// TIA Portal project "tasl1" (V16)
// Vorlageprojekt für das Buch mit Zielsystem S7-1200

(* hardware
DEVICE "S7-1200-Station_1"  S7-1200 Station
   slot 0: "Baugruppenträger_0"  Rack  V1.0
   slot 1: "PLC_1"  CPU 1211C DC/DC/DC  6ES7 211-1AE40-0XB0  V4.1
*)

// ===== PLC "PLC_1"  CPU 1211C DC/DC/DC =====

VAR_GLOBAL   // PLC tag table "Standard-Variablentabelle"
   "Tag_1" AT %A0.0 : Bool;
   "Tag_2" AT %E0.0 : Bool;
   "Tag_3" AT %E0.1 : Bool;
   "start" AT %I10.0 : Bool;
   "conv6" AT %Q10.0 : Bool;
   "stop" AT %I10.1 : Bool;
   "Tag_7" AT %I10.2 : Bool;
   "pusher" AT %Q10.2 : Bool;
   "Tag_9" AT %M0.0 : Bool;
   "x" AT %M0.1 : Bool;
   "front" AT %I10.4 : Bool;
   "back" AT %I10.3 : Bool;
   "conv2" AT %Q10.1 : Bool;
   "back(1)" AT %I10.3 : Bool;
END_VAR

// folder: System blocks/Program resources

DATA_BLOCK "time"   // DB1
{ S7_Optimized_Access := 'TRUE' }
AUTHOR : Simatic
FAMILY : IEC
NAME : IEC_TMR
VERSION : 1.0
// stored: InstanceOfName IEC_TIMER
"IEC_TIMER"
BEGIN
END_DATA_BLOCK

// folder: (top level)

FUNCTION "MHJ-PLC-Lab-Function-S71200" : Void   // FC9000, SCL
{ S7_Optimized_Access := 'TRUE' }
VERSION : 0.1
   VAR_TEMP
      rdTimeReturn : Int;
      outputTime : DTL;
      SyncVal : Byte;
      forVal : Int;
      forVal_2 : Int;
      Value : Byte;
   END_VAR
   VAR CONSTANT
      CompVal : Byte := 16#34;
      Value_01 : Byte := 16#11;
      Value_01_DW : DWord := 16#A165_D992;
      Value_02_DW : DWord := 16#58BE_4401;
   END_VAR
BEGIN

   #Value:=PEEK(area := 16#82,
        dbNumber := 0,
        byteOffset := 511);
   #Value := #Value + 1;

   POKE(area := 16#82,
        dbNumber := 0,
        byteOffset := 511,
        value := #Value);

   POKE(area:=16#81,
        dbNumber:=0,
        byteOffset:=1016,
        value:=#Value_01_DW);
   POKE(area := 16#81,
        dbNumber := 0,
        byteOffset := 1020,
        value := #Value_02_DW);

   POKE(area := 16#81,
        dbNumber := 0,
        byteOffset := 511,
        value := B#16#00);

   FOR #forVal := 0 TO 120 DO
       FOR #forVal_2:=0 TO 10 DO
           #rdTimeReturn:=RD_SYS_T(#outputTime);
           #rdTimeReturn := WR_SYS_T(#outputTime);
           #rdTimeReturn := RD_SYS_T(#outputTime);
           #rdTimeReturn := WR_SYS_T(#outputTime);
       END_FOR;
       #SyncVal:= PEEK(area := 16#81,
                      dbNumber := 0,
                      byteOffset := 511);
       IF #SyncVal = #CompVal THEN
          GOTO M_1;
       END_IF;
   END_FOR;
   RETURN;

   M_1:
   POKE(area := 16#81,
        dbNumber := 0,
        byteOffset := 511,
        value := B#16#0);
END_FUNCTION

ORGANIZATION_BLOCK "Main"   // OB1, LAD, ProgramCycle
TITLE = "Main Program Sweep (Cycle)"
{ S7_Optimized_Access := 'TRUE' }
VERSION : 0.1
   VAR_INPUT
      Initial_Call : Bool;   // Initial call of this OB
      Remanence : Bool;   // =True, if remanent data are available
   END_VAR
   VAR_TEMP   // added for the SCL form of the ladder/FBD networks
      _w1 : Bool;
   END_VAR
BEGIN

REGION Network 1: Konnektierungsbaustein für PLC-Lab
   // Im Netzwerk 1 wird der Konnektierungsbaustein für PLC-Lab aufgerufen.
   // Dieser Aufruf darf nicht entfernt werden!
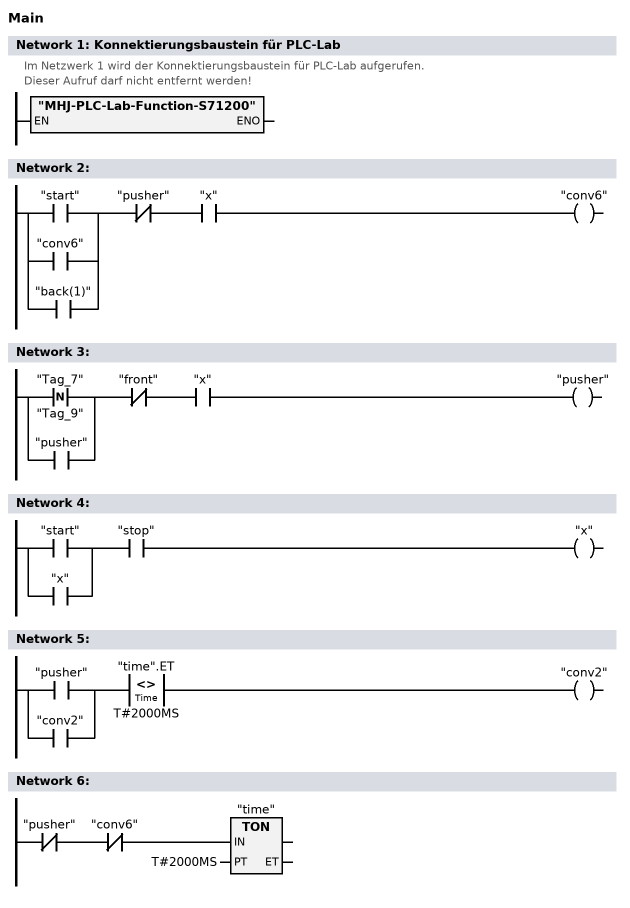
   RUNG wire#powerrail
      "MHJ-PLC-Lab-Function-S71200"()
   END_RUNG
   // the same network as SCL:
   "MHJ-PLC-Lab-Function-S71200"();
END_REGION

REGION Network 2
   RUNG wire#powerrail
      Contact( "start" )
      wire#w1
      I_Contact( "pusher" )
      Contact( "x" )
      Coil( "conv6" )
   END_RUNG
   RUNG wire#powerrail
      Contact( "conv6" )
   END_RUNG wire#w1
   RUNG wire#powerrail
      Contact( "back(1)" )
   END_RUNG wire#w1
   // the same network as SCL:
   "conv6" := ("start" OR "conv6" OR "back(1)") AND NOT "pusher" AND "x";
END_REGION

REGION Network 3
   RUNG wire#powerrail
      N_Contact(operand := "Tag_7", bit := "Tag_9")
      wire#w1
      I_Contact( "front" )
      Contact( "x" )
      Coil( "pusher" )
   END_RUNG
   RUNG wire#powerrail
      Contact( "pusher" )
   END_RUNG wire#w1
   // the same network as SCL:
   #_w1 := NOT "Tag_7" AND "Tag_9";   // falling edge of "Tag_7"
   "Tag_9" := "Tag_7";
   "pusher" := (#_w1 OR "pusher") AND NOT "front" AND "x";
END_REGION

REGION Network 4
   RUNG wire#powerrail
      Contact( "start" )
      wire#w1
      Contact( "stop" )
      Coil( "x" )
   END_RUNG
   RUNG wire#powerrail
      Contact( "x" )
   END_RUNG wire#w1
   // the same network as SCL:
   "x" := ("start" OR "x") AND "stop";
END_REGION

REGION Network 5
   RUNG wire#powerrail
      Contact( "pusher" )
      wire#w1
      { S7_Templates := "SrcType := Time" } NE_Contact(in1 := "time".ET, in2 := T#2000MS)
      Coil( "conv2" )
   END_RUNG
   RUNG wire#powerrail
      Contact( "conv2" )
   END_RUNG wire#w1
   // the same network as SCL:
   "conv2" := ("pusher" OR "conv2") AND ("time".ET <> T#2000MS);
END_REGION

REGION Network 6
   "time".TON(IN := NOT "pusher" AND NOT "conv6", PT := T#2000MS);
END_REGION
END_ORGANIZATION_BLOCK